TYPE ST_TestSuiteInstance :
STRUCT
    eTestSuiteRunState : E_TestSuiteRunState := E_TestSuiteRunState.IDLE;
END_STRUCT
END_TYPE

(* stored: Version 1.1.0.1, ProductVersion 3.1.4022.12
   DUT ST_TestSuiteInstance: Id {016951be-9167-42bd-ae10-8e1a68d8330a} *)
